(* IEC 61131-3 sources: AXOpen/src/TestSandbox/ctrl/src/TestedControlUnit, 3 files *)

(* ---- IdGenerator.st ---- *)
NAMESPACE sandboxtest.StandardControlUnit
    USING AXOpen.Core;
    USING System.Strings;
    USING AXOpen.Cognex.Vision.v_6_0_0_0;
    USING AXOpen.Elements;

    // just prepared but not used -> reason -> Exist task not exist yet
    INTERFACE PUBLIC ITestIdGenerator
        METHOD GetSize : Int
        END_METHOD
        METHOD Increment : BOOL
        END_METHOD
        METHOD GetRootRecordName : STRING
        END_METHOD
        METHOD GetNext : STRING
        END_METHOD
        METHOD InitializeWithPrefix
            VAR_INPUT
                Prefix : STRING;
            END_VAR
        END_METHOD
    END_INTERFACE

    {#ix-attr:[RenderIgnore()]}
    CLASS PUBLIC TestIdGenerator
        EXTENDS AXOpen.Core.AxoObject
        IMPLEMENTS ITestIdGenerator
        // VAR  CONSTANT PUBLIC
        //     {#ix-attr:[RenderIgnore()]}
        //     MAX_SIZE : INT := 1000; (* Comment *)
        //     {#ix-attr:[RenderIgnore()]}
        //     ROOT_RECORD_NAME : STRING := 'process_set'; (* Comment *)
        // END_VAR
        VAR
            {#ix-attr:[RenderIgnore()]}
            _Names : ARRAY[0..10] OF STRING;
            CurrentIndex : INT;
            LastId : STRING;
        END_VAR

        METHOD PUBLIC GetNext : STRING
            IF CurrentIndex < 0 THEN
                CurrentIndex := 0;
            END_IF;
            IF CurrentIndex > 10 THEN
                CurrentIndex := 0;
            END_IF;
            LastId := _Names[CurrentIndex];
            GetNext := LastId;
        END_METHOD

        METHOD PUBLIC Increment : BOOL
            CurrentIndex := CurrentIndex + 1;
            Increment := CurrentIndex <= 10;
        END_METHOD

        METHOD PUBLIC GetSize : INT
            GetSize := 10;
        END_METHOD

        METHOD PUBLIC GetRootRecordName : STRING
            GetRootRecordName := 'process_set';
        END_METHOD

        METHOD PUBLIC InitializeWithPrefix
            VAR_INPUT
                Prefix : STRING;
            END_VAR
            VAR
                index : INT := 0; (* LOCAL INDEX *)
            END_VAR
            THIS.CurrentIndex := 0;
            FOR index := 0 TO 10 BY 1 DO
                _Names[index] := Concat(Prefix, '_', ToString(index));
            END_FOR;
        END_METHOD
    END_CLASS

END_NAMESPACE

(* ---- CuComponents.st ---- *)
NAMESPACE sandboxtest.StandardControlUnit
    USING AXOpen.Core;
    USING System.Strings;
    USING AXOpen.Cognex.Vision.v_6_0_0_0;

    ///<summary>
    /// Groups components of this controller unit.
    ///</summary>
    CLASS Components
        EXTENDS AXOpen.Core.AxoObject
        VAR PUBLIC
            counter : INT;
            {#ix-attr:[Container(Layout.Tabs)]}
           // HERE DECLARE COMPONENTS USED BY THIS CONTROLLED UNIT
            Cylinder_0 : AXOpen.Components.Pneumatics.AxoCylinder;
            Cylinder_1 : AXOpen.Components.Pneumatics.AxoCylinder;
            Cylinder_2 : AXOpen.Components.Pneumatics.AxoCylinder;
            Cylinder_3 : AXOpen.Components.Pneumatics.AxoCylinder;
            Cylinder_4 : AXOpen.Components.Pneumatics.AxoCylinder;
            Cylinder_5 : AXOpen.Components.Pneumatics.AxoCylinder;
            Cylinder_6 : AXOpen.Components.Pneumatics.AxoCylinder;
            Cylinder_7 : AXOpen.Components.Pneumatics.AxoCylinder;
            Cylinder_8 : AXOpen.Components.Pneumatics.AxoCylinder;
            Cylinder_9 : AXOpen.Components.Pneumatics.AxoCylinder;
            Camera_0 : AXOpen.Cognex.Vision.v_6_0_0_0.AxoInsight;
            Camera_1 : AXOpen.Cognex.Vision.v_6_0_0_0.AxoInsight;
            Reader_0 : AXOpen.Cognex.Vision.v_6_0_0_0.AxoDataman;
            Reader_1 : AXOpen.Cognex.Vision.v_6_0_0_0.AxoDataman;
        END_VAR

        METHOD PUBLIC Update
            VAR_INPUT
                parent : IAxoObject;
            END_VAR
            VAR_INPUT
                Inputs : REF_TO sandboxtest.Inputs;
                Outputs : REF_TO sandboxtest.Outputs;
            END_VAR
            THIS.Initialize(parent);
            // HERE INITIALIZE YOUR COMPONENTS
            Cylinder_0.Run(THIS, Inputs^.B0[0], Inputs^.B0[1], Outputs^.B0[2], Outputs^.B0[3]);
            Cylinder_1.Run(THIS, Inputs^.B1[0], Inputs^.B1[1], Outputs^.B1[2], Outputs^.B1[3]);
            Cylinder_2.Run(THIS, Inputs^.B2[0], Inputs^.B2[1], Outputs^.B2[2], Outputs^.B2[3]);
            Cylinder_3.Run(THIS, Inputs^.B3[0], Inputs^.B3[1], Outputs^.B3[2], Outputs^.B3[3]);
            Cylinder_4.Run(THIS, Inputs^.B4[0], Inputs^.B4[1], Outputs^.B4[2], Outputs^.B4[3]);
            Cylinder_5.Run(THIS, Inputs^.B5[0], Inputs^.B5[1], Outputs^.B5[2], Outputs^.B5[3]);
            Cylinder_6.Run(THIS, Inputs^.B6[0], Inputs^.B6[1], Outputs^.B6[2], Outputs^.B6[3]);
            Cylinder_7.Run(THIS, Inputs^.B7[0], Inputs^.B7[1], Outputs^.B7[2], Outputs^.B7[3]);
            Cylinder_8.Run(THIS, Inputs^.B8[0], Inputs^.B8[1], Outputs^.B8[2], Outputs^.B8[3]);
            Cylinder_9.Run(THIS, Inputs^.B9[0], Inputs^.B9[1], Outputs^.B9[2], Outputs^.B9[3]);

            Reader_0.Run( parent            :=  THIS,
                refAcquisitionStatus        :=  REF(Inputs^._Reader_0_Acquisition_Status_1),
                refSoftEventStatus          :=  REF(Inputs^._Reader_0_Soft_Event_Control_1),
                refResultsStatus            :=  REF(Inputs^._Reader_0_Results_Status_1),
                refResultData               :=  REF(Inputs^._Reader_0_Result_Data_128_bytes_1),
                refUserData                 :=  REF(Outputs^._Reader_0_User_Data_128_bytes_1),
                refAcquisitionControl       :=  REF(Outputs^._Reader_0_Acquisition_Control_1),
                refResultsControl           :=  REF(Outputs^._Reader_0_Results_Control_1),
                refSoftEventControl         :=  REF(Outputs^._Reader_0_Soft_Event_Control_1)
            );

            Reader_1.Run( parent            :=  THIS,
                refAcquisitionStatus        :=  REF(Inputs^._Reader_1_Acquisition_Status_1),
                refSoftEventStatus          :=  REF(Inputs^._Reader_1_Soft_Event_Control_1),
                refResultsStatus            :=  REF(Inputs^._Reader_1_Results_Status_1),
                refResultData               :=  REF(Inputs^._Reader_1_Result_Data_128_bytes_1),
                refUserData                 :=  REF(Outputs^._Reader_1_User_Data_128_bytes_1),
                refAcquisitionControl       :=  REF(Outputs^._Reader_1_Acquisition_Control_1),
                refResultsControl           :=  REF(Outputs^._Reader_1_Results_Control_1),
                refSoftEventControl         :=  REF(Outputs^._Reader_1_Soft_Event_Control_1)
            );

            Camera_0.Run(  parent                  :=  THIS,
                            refAcquisitionStatus    :=  REF(Inputs^ ._Camera_0_Acquisition_Status_1),
                            refInspectionStatus     :=  REF(Inputs^ ._Camera_0_Inspection_Status_1),
                            refCommandStatus        :=  REF(Inputs^ ._Camera_0_Command_Control_1),
                            refSoftEventStatus      :=  REF(Inputs^ ._Camera_0_SoftEvent_Control_1),
                            refResultData           :=  REF(Inputs^ ._Camera_0_Results_64_bytes_1),
                            refInspectionControl    :=  REF(Outputs^._Camera_0_Inspection_Control_1),
                            refCommandControl       :=  REF(Outputs^._Camera_0_Command_Control_1),
                            refAcquisitionControl   :=  REF(Outputs^._Camera_0_Acquisition_Control_1),
                            refSoftEventControl     :=  REF(Outputs^._Camera_0_SoftEvent_Control_1),
                            refUserData             :=  REF(Outputs^._Camera_0_User_Data_64_bytes_1));

            Camera_1.Run(  parent                  :=  THIS,
                            refAcquisitionStatus    :=  REF(Inputs^ ._Camera_1_Acquisition_Status_1),
                            refInspectionStatus     :=  REF(Inputs^ ._Camera_1_Inspection_Status_1),
                            refCommandStatus        :=  REF(Inputs^ ._Camera_1_Command_Control_1),
                            refSoftEventStatus      :=  REF(Inputs^ ._Camera_1_SoftEvent_Control_1),
                            refResultData           :=  REF(Inputs^ ._Camera_1_Results_64_bytes_1),
                            refInspectionControl    :=  REF(Outputs^._Camera_1_Inspection_Control_1),
                            refCommandControl       :=  REF(Outputs^._Camera_1_Command_Control_1),
                            refAcquisitionControl   :=  REF(Outputs^._Camera_1_Acquisition_Control_1),
                            refSoftEventControl     :=  REF(Outputs^._Camera_1_SoftEvent_Control_1),
                            refUserData             :=  REF(Outputs^._Camera_1_User_Data_64_bytes_1));
                          ;
        END_METHOD
    END_CLASS

END_NAMESPACE

(* ---- StandardCu.st ---- *)
NAMESPACE sandboxtest.StandardControlUnit
    USING AXOpen.Core;
    USING System.Strings;
    USING AXOpen.Cognex.Vision.v_6_0_0_0;

    ///<summary>
    /// Represents controlled units and high level task coordination.
    ///</summary>
    CLASS CU
        EXTENDS AXOpen.Core.AxoObject
        VAR PUBLIC
            ///<summary>
            /// Handles and intializes components used by this unit.
            ///</summary>
            Components : Components;
            ///<summary>
            /// Ground sequence. Contains logic that brings the unit into initial state.
            ///</summary>
            GroundSequence : GroundSequence;
            ///<summary>
            /// Automatic sequence. Contains logic for automatic operations of this unit.
            ///</summary>
            AutomatSequence : AutomatSequence;
            ///<summary>
            /// Service mode contains logic for service/manual operations.
            ///</summary>
            ServiceMode : ServiceMode;
            StationName : STRING;
            SettingSourceManager : AXOpen.DATA.IAxoDataExchange;
            SettingSourceData : REF_TO FragmentProcessData;
            ProcessData : REF_TO ProcessDataManger;
        END_VAR

        METHOD PUBLIC InvokeMode : INT
            VAR_INPUT
                iMode : INT;
            END_VAR
            ;
            InvokeMode := 0;
            CASE iMode OF
                10:
                    AutomatSequence.Invoke();
                    IF AutomatSequence.IsBusy() THEN
                        InvokeMode := iMode;
                    END_IF;
                20:
                    GroundSequence.Invoke();
                    IF GroundSequence.IsDone() THEN
                        InvokeMode := iMode;
                    END_IF;
                30:
                    ServiceMode.Invoke();
                    IF ServiceMode.IsBusy() THEN
                        InvokeMode := iMode;
                    END_IF;
            END_CASE;
        END_METHOD
        ///<summary>
        /// Runs this unit.
        ///</summary>

        METHOD PUBLIC Run
            VAR_INPUT
                _parent : AXOpen.Core.IAxoContext;
                _stationName : STRING;
                _settingSourceManager : AXOpen.DATA.IAxoDataExchange;
                _settingSourceData : REF_TO FragmentProcessData;
                Inputs : REF_TO sandboxtest.Inputs;
                Outputs : REF_TO sandboxtest.Outputs;
            END_VAR
            StationName := _stationName;
            SettingSourceManager := _settingSourceManager;
            SettingSourceData := _settingSourceData;
            THIS.Initialize(_parent);
            THIS.Execute(Inputs, Outputs);
        END_METHOD

        METHOD PRIVATE Execute
            VAR_INPUT
                Inputs : REF_TO sandboxtest.Inputs;
                Outputs : REF_TO sandboxtest.Outputs;
            END_VAR
            // Component I/O immange and management handling.
            Components.Update(THIS, Inputs, Outputs);
            // Process data manager
            ProcessData^.Run(THIS);
            // Handles ground sequence
            GroundSequence.Run(THIS, REF(Components), ProcessData, SettingSourceData, SettingSourceManager);
            // Restores other states when Ground executes
            IF (GroundSequence.IsBusy()) THEN
                AutomatSequence.Restore();
                ServiceMode.Restore();
            END_IF;
            // Handles automatic sequence (ground must be previously done)
            AutomatSequence.IsDisabled := GroundSequence.Status <> eAxoTaskState#Done;
            AutomatSequence.Run(THIS, REF(Components), ProcessData, SettingSourceData, SettingSourceManager, REF(StationName));
            // Handles service/manual mode
            ServiceMode.Run(THIS, Components);
            IF ServiceMode.IsBusy() THEN
                GroundSequence.Restore();
                AutomatSequence.Restore();
            END_IF;
        END_METHOD
    END_CLASS

END_NAMESPACE
